TYPE U_XTS_STATION_STATE :
UNION
  stState             : ARRAY[1..MAX_STATION] OF ST_STATION_STATE;

  byState   AT %Q*    : ARRAY[1..MAX_STATION] OF
                        ARRAY[1..SIZEOF(ST_STATION_STATE)] OF BYTE;
END_UNION
END_TYPE

(* stored: Version 1.1.0.1, ProductVersion 3.1.4026.13
   DUT U_XTS_STATION_STATE: Id {7b8a9ba5-33f2-4709-9d50-2b02a37bb6a5} *)
